// Mitsubishi GX Works2 project: onwork_noon   PLC: FX3G

// global labels: Global1
VAR_GLOBAL
  start_machineA AT X010 : BOOL;
  Touch_Sen AT M1 : BOOL;
  stop_machineA AT X005 : BOOL;
  Sen_Camera AT M2 : BOOL;
  Sen_30 AT X001 : BOOL;
  Ziluf_on AT Y004 : BOOL;
  Sen_15 AT X002 : BOOL;
  helpA AT M3 : BOOL;
  REG_InvetoryBiscuits AT D1102 : REAL;
END_VAR
VAR_GLOBAL CONSTANT
  Const_Biscuits : REAL := 6;
END_VAR
VAR_GLOBAL
  REG_Ziluf AT D1110 : REAL;
  REG_InvetoryCream AT D1104 : REAL;
END_VAR
VAR_GLOBAL CONSTANT
  Const_Cream : REAL := 300;
  Const_Zero : REAL;
  Const_InitInventoryBiscuits : REAL := 12;
  Const_InitInventoryCream : REAL := 600;
END_VAR
VAR_GLOBAL
  Sw_7_StartDay AT X007 : BOOL;
  M_TurnOffAll AT M7 : BOOL;
  Li_7_Day AT Y007 : BOOL;
  M_StartBlinking AT M8 : BOOL;
  Light_Generator AT M9 : BOOL;
  TC_BLINK_1 AT TC1 : BOOL;
  TS_BLINK_1 AT TS1 : BOOL;
  M_Blinking_Light1 AT M200 : BOOL;
  TC_BLINK_2 AT TC2 : BOOL;
END_VAR
VAR_GLOBAL CONSTANT
  CONSTANT3_word : INT := 3;
END_VAR
VAR_GLOBAL
  TS_BLINK_2 AT TS2 : BOOL;
  M_Blinking_Light2 AT M201 : BOOL;
  REG_InvetoryChocolate AT D1106 : REAL;
END_VAR
VAR_GLOBAL CONSTANT
  Const_Chocolate : REAL := 240;
END_VAR
VAR_GLOBAL
  M_InvetoryBiscuits AT M10 : BOOL;
  M_InvetoryCream AT M11 : BOOL;
  M_InvetoryChocolate AT M12 : BOOL;
  M_canStartDay AT M13 : BOOL;
  Current_in_process AT D1118 : REAL;
  Ziluf_timer AT TC0 : BOOL;
  TimerZiluf AT TC3 : BOOL;
END_VAR
VAR_GLOBAL CONSTANT
  TwoSeconds : INT := 20;
  SixSeconds : INT := 60;
END_VAR
VAR_GLOBAL
  TC_Shinua AT TC5 : BOOL;
END_VAR
VAR_GLOBAL CONSTANT
  FourSeconds : INT := 40;
END_VAR
VAR_GLOBAL
  TS_Shinua AT TS5 : BOOL;
  Sw_CreamToZiluf AT X011 : BOOL;
  TS_Ziluf AT TS3 : BOOL;
  TransportLight0 AT Y000 : BOOL;
  TrS1 AT Y001 : BOOL;
  TC_CloseDayTimer AT TC12 : BOOL;
END_VAR
VAR_GLOBAL CONSTANT
  ThreeSeconds : INT := 30;
END_VAR
VAR_GLOBAL
  TS_CloseDayTimer AT TS12 : BOOL;
  Ziluf_is_empty AT M22 : BOOL;
  Current_is_empty AT M24 : BOOL;
  Ziluf_is_full AT M23 : BOOL;
END_VAR
VAR_GLOBAL CONSTANT
  Const_CreamInit : REAL := 600;
  Const_ChocolateInit : REAL := 1000;
  Const_BiscuitsInit : REAL := 20;
END_VAR
VAR_GLOBAL
  input_pulse AT X006 : BOOL;
  analon_input_1 AT D8280 : INT;
  analog_input_val AT D1150 : REAL;
END_VAR
VAR_GLOBAL CONSTANT
  val1_analog_input_1 : REAL := 419;
END_VAR
VAR_GLOBAL
  frosting_type AT D4000 : REAL;
END_VAR
VAR_GLOBAL CONSTANT
  val1 : REAL := 1;
END_VAR
VAR_GLOBAL
  greater_than_1 AT M20 : BOOL;
END_VAR
VAR_GLOBAL CONSTANT
  val5 : REAL := 5;
END_VAR
VAR_GLOBAL
  less_than_5 AT M57 : BOOL;
  in_process AT TS7 : BOOL;
  double_frosting AT M32 : BOOL;
  regular_frosting AT M30 : BOOL;
END_VAR
VAR_GLOBAL CONSTANT
  val6 : REAL := 6;
END_VAR
VAR_GLOBAL
  greater_than_6 AT M25 : BOOL;
END_VAR
VAR_GLOBAL CONSTANT
  val10 : REAL := 10;
END_VAR
VAR_GLOBAL
  less_than_10 AT M27 : BOOL;
END_VAR
VAR_GLOBAL CONSTANT
  val120 : REAL := 120;
END_VAR
VAR_GLOBAL
  REG_immersion_tank AT D6500 : REAL;
END_VAR
VAR_GLOBAL CONSTANT
  val240 : REAL := 240;
END_VAR
VAR_GLOBAL
  frosting_timer AT TC7 : BOOL;
END_VAR
VAR_GLOBAL CONSTANT
  val0 : REAL;
  five_sec : INT := 5;
END_VAR
VAR_GLOBAL
  frosting_light AT Y003 : BOOL;
  error AT Y005 : BOOL;
  REG_CHECK AT D7000 : REAL;
  TimerZiluf_indicator AT TS3 : BOOL;
  pack_krembo AT X000 : BOOL;
  REG_done_indevidual_k_platform AT D3002 : REAL;
  almost_done_packing_platform AT Y002 : BOOL;
  REG_done_krembo_total AT D2222 : REAL;
END_VAR
VAR_GLOBAL CONSTANT
  const40 : REAL := 40;
END_VAR
VAR_GLOBAL
  VALUE_OUTPUT_ANALOG AT D2121 : REAL;
  value_analog_show_screen_REALLY AT D8282 : INT;
  done3 AT M14 : BOOL;
  start_pack AT M40 : BOOL;
  light_timer2_off AT TS2 : BOOL;
  light_timer1_off AT TS1 : BOOL;
  end_successfully AT M15 : BOOL;
  done4 AT M39 : BOOL;
  added_done_packed AT M45 : BOOL;
  timer_reset AT M42 : BOOL;
  light_counter AT CC10 : BOOL;
END_VAR
VAR_GLOBAL CONSTANT
  val3 : INT := 3;
END_VAR
VAR_GLOBAL
  light_counter_val AT CN10 : INT;
  need_flash AT M35 : BOOL;
END_VAR
VAR_GLOBAL CONSTANT
  val1_word : INT := 1;
END_VAR
VAR_GLOBAL
  supply_end AT M21 : BOOL;
  blink_end1 AT M47 : BOOL;
  no_supply_timer AT TC9 : BOOL;
END_VAR
VAR_GLOBAL CONSTANT
  three_sec : INT := 30;
END_VAR
VAR_GLOBAL
  TS_nosupply_timer AT TS9 : BOOL;
  M49_Y7 AT M49 : BOOL;
  tm_nosupply2 AT TC11 : BOOL;
  TS2_nosup AT TS11 : BOOL;
  M51_offM49 AT M51 : BOOL;
  final_tm AT TC15 : BOOL;
  final_tm_indecator AT TS15 : BOOL;
  blink_indecator AT M55 : BOOL;
END_VAR
VAR_GLOBAL CONSTANT
  five_sec_frosting : INT := 50;
END_VAR
VAR_GLOBAL
  not_enough_krembo AT M13 : BOOL;
END_VAR

// task Task_01 (event TRUE, interval 0, priority 31): POU_01

PROGRAM POU_01
VAR
  TransportLight1 : BOOL;
END_VAR
(* structured ladder/FBD written out as ST: instructions are called as NAME(EN, inputs, outputs); _pN, _eN, _tN stand for wires *)
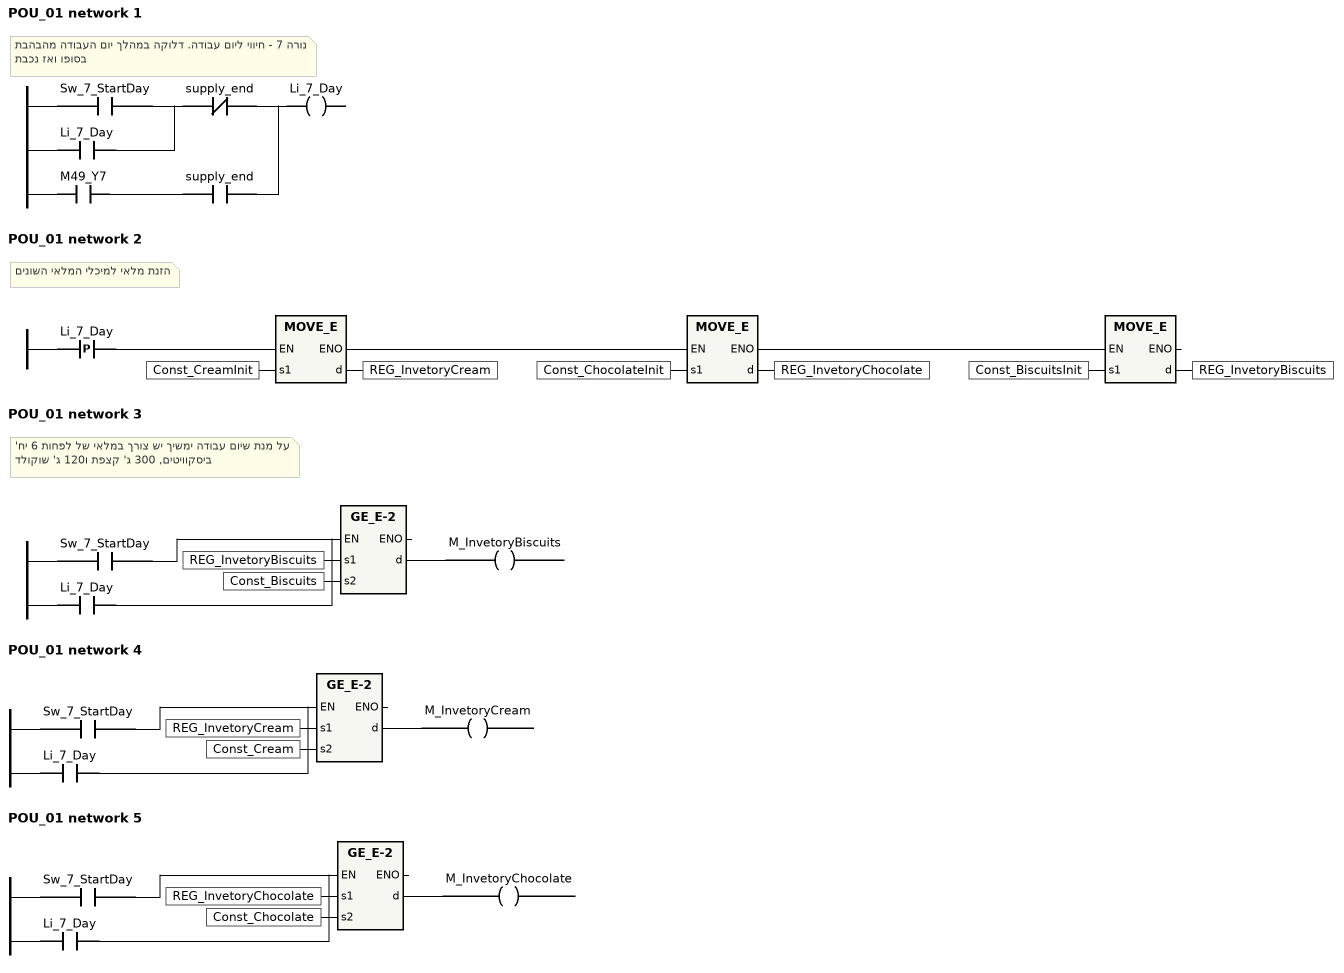
(* network 1 *)
(* נורה 7 - חיווי ליום עבודה. דלוקה במהלך יום העבודה מהבהבת בסופו ואז נכבת *)
Li_7_Day := ((Sw_7_StartDay OR Li_7_Day) AND NOT supply_end) OR (M49_Y7 AND supply_end);
(* network 2 *)
(* הזנת מלאי למיכלי המלאי השונים *)
_e1 := MOVE_E(LDP(TRUE, Li_7_Day), Const_CreamInit, REG_InvetoryCream);
_e2 := MOVE_E(_e1, Const_ChocolateInit, REG_InvetoryChocolate);
MOVE_E(_e2, Const_BiscuitsInit, REG_InvetoryBiscuits);
(* network 3 *)
(* על מנת שיום עבודה ימשיך יש צורך במלאי של לפחות 6 יח' ביסקוויטים, 300 ג' קצפת ו120 ג' שוקולד *)
GE_E(Sw_7_StartDay OR Li_7_Day, REG_InvetoryBiscuits, Const_Biscuits, _t1);
M_InvetoryBiscuits := _t1;
(* network 4 *)
GE_E(Sw_7_StartDay OR Li_7_Day, REG_InvetoryCream, Const_Cream, _t1);
M_InvetoryCream := _t1;
(* network 5 *)
GE_E(Sw_7_StartDay OR Li_7_Day, REG_InvetoryChocolate, Const_Chocolate, _t1);
M_InvetoryChocolate := _t1;
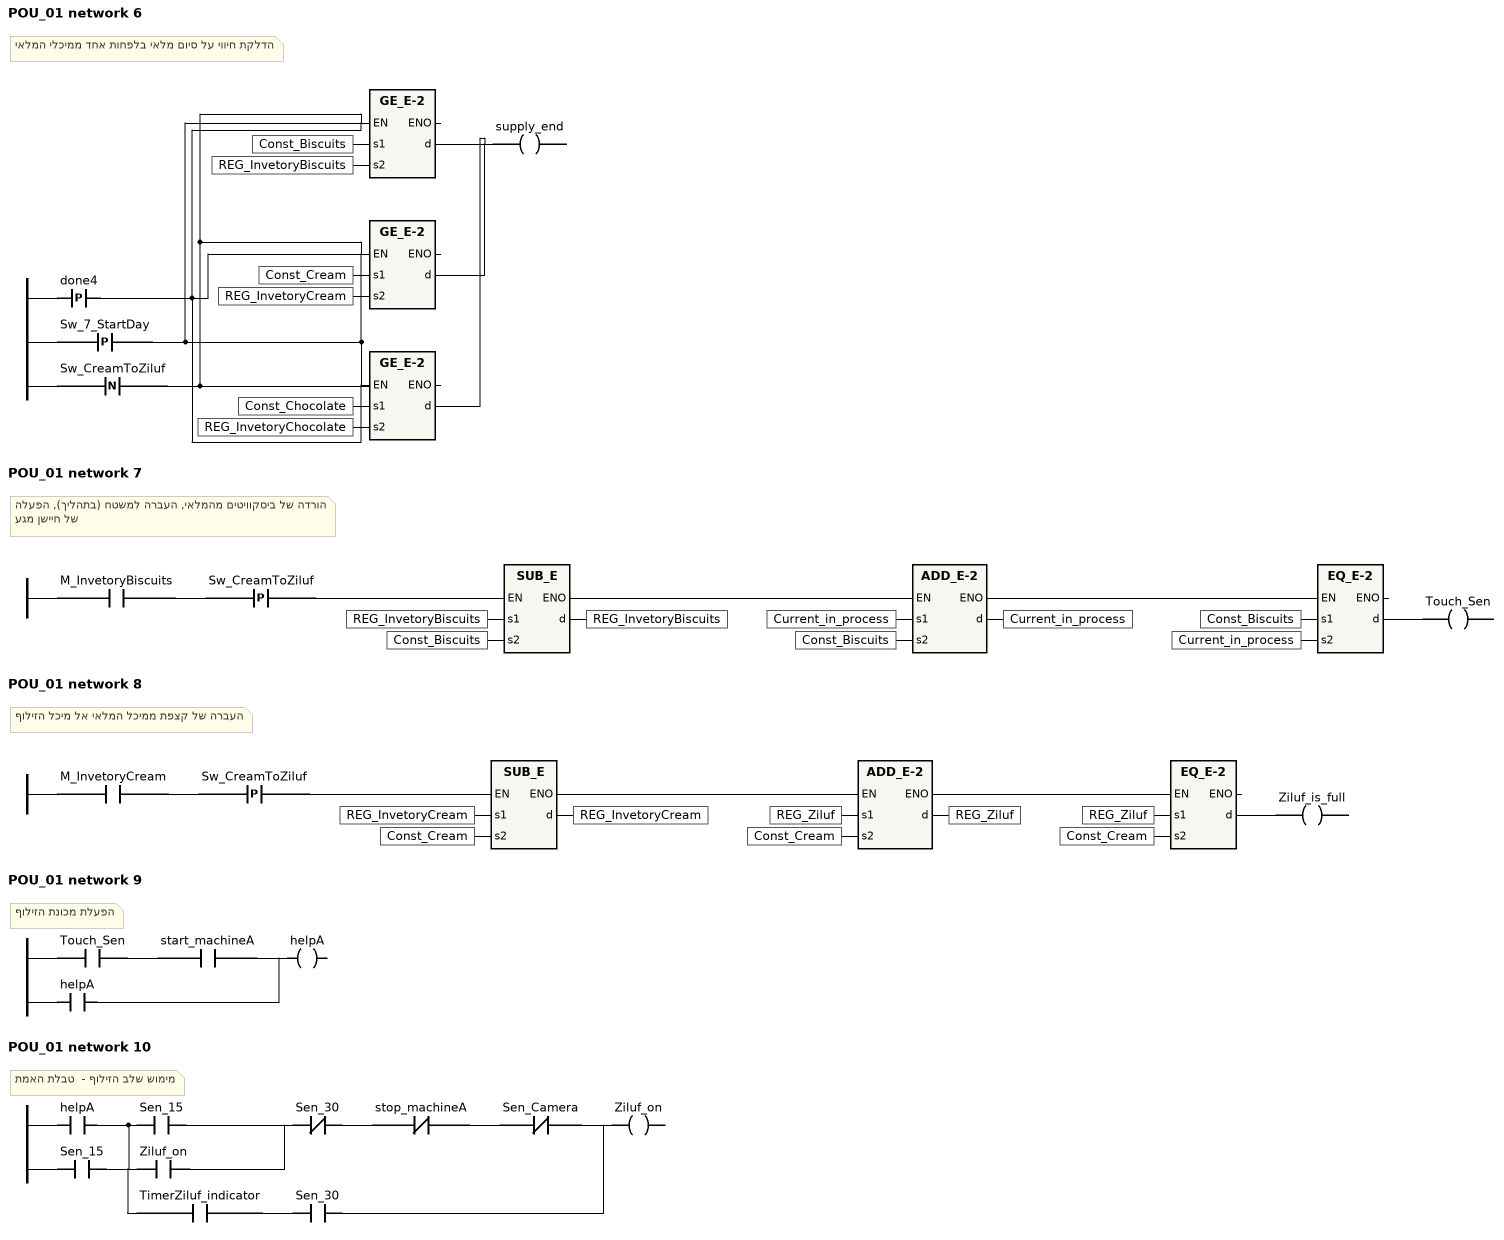
(* network 6 *)
(* הדלקת חיווי על סיום מלאי בלפחות אחד ממיכלי המלאי *)
_p1 := LDP(TRUE, done4) OR LDP(TRUE, Sw_7_StartDay) OR LDF(TRUE, Sw_CreamToZiluf);
GE_E(_p1, Const_Biscuits, REG_InvetoryBiscuits, _t2);
GE_E(_p1, Const_Cream, REG_InvetoryCream, _t3);
GE_E(_p1, Const_Chocolate, REG_InvetoryChocolate, _t4);
supply_end := _t2 OR _t3 OR _t4;
(* network 7 *)
(* הורדה של ביסקוויטים מהמלאי, העברה למשטח (בתהליך), הפעלה של חיישן מגע *)
_e1 := SUB_E(M_InvetoryBiscuits AND LDP(TRUE, Sw_CreamToZiluf), REG_InvetoryBiscuits, Const_Biscuits, REG_InvetoryBiscuits);
_e2 := ADD_E(_e1, Current_in_process, Const_Biscuits, Current_in_process);
EQ_E(_e2, Const_Biscuits, Current_in_process, _t3);
Touch_Sen := _t3;
(* network 8 *)
(* העברה של קצפת ממיכל המלאי אל מיכל הזילוף *)
_e1 := SUB_E(M_InvetoryCream AND LDP(TRUE, Sw_CreamToZiluf), REG_InvetoryCream, Const_Cream, REG_InvetoryCream);
_e2 := ADD_E(_e1, REG_Ziluf, Const_Cream, REG_Ziluf);
EQ_E(_e2, REG_Ziluf, Const_Cream, _t3);
Ziluf_is_full := _t3;
(* network 9 *)
(* הפעלת מכונת הזילוף *)
helpA := (Touch_Sen AND start_machineA) OR helpA;
(* network 10 *)
(* מימוש שלב הזילוף -  טבלת האמת *)
Ziluf_on := (((((helpA AND Sen_15) OR (helpA AND Ziluf_on)) AND NOT Sen_30) AND NOT stop_machineA) AND NOT Sen_Camera) OR (Sen_15 AND TimerZiluf_indicator AND Sen_30);
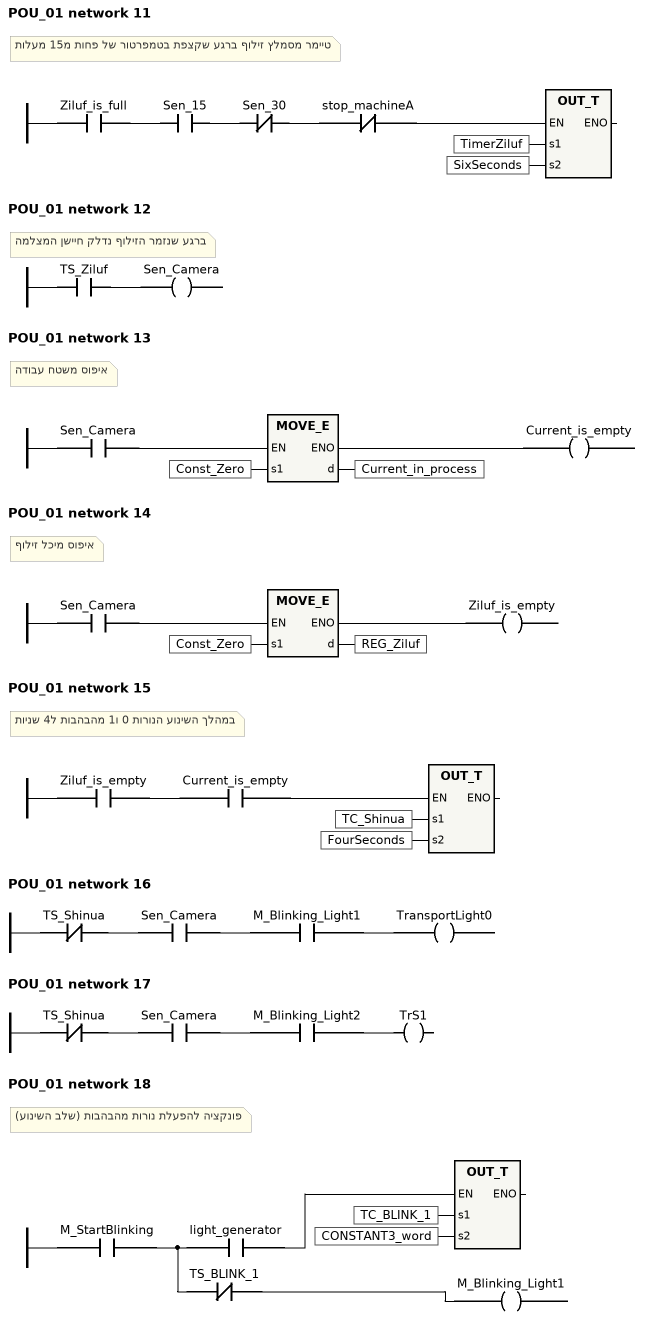
(* network 11 *)
(* טיימר מסמלץ זילוף ברגע שקצפת בטמפרטור של פחות מ15 מעלות *)
OUT_T(Ziluf_is_full AND Sen_15 AND NOT Sen_30 AND NOT stop_machineA, TimerZiluf, SixSeconds);
(* network 12 *)
(* ברגע שנזמר הזילוף נדלק חיישן המצלמה *)
Sen_Camera := TS_Ziluf;
(* network 13 *)
(* איפוס משטח עבודה *)
_e1 := MOVE_E(Sen_Camera, Const_Zero, Current_in_process);
Current_is_empty := _e1;
(* network 14 *)
(* איפוס מיכל זילוף *)
_e1 := MOVE_E(Sen_Camera, Const_Zero, REG_Ziluf);
Ziluf_is_empty := _e1;
(* network 15 *)
(* במהלך השינוע הנורות 0 ו1 מהבהבות ל4 שניות *)
OUT_T(Ziluf_is_empty AND Current_is_empty, TC_Shinua, FourSeconds);
(* network 16 *)
TransportLight0 := NOT TS_Shinua AND Sen_Camera AND M_Blinking_Light1;
(* network 17 *)
TrS1 := NOT TS_Shinua AND Sen_Camera AND M_Blinking_Light2;
(* network 18 *)
(* פונקציה להפעלת נורות מהבהבות (שלב השינוע) *)
OUT_T(M_StartBlinking AND light_generator, TC_BLINK_1, CONSTANT3_word);
M_Blinking_Light1 := M_StartBlinking AND NOT TS_BLINK_1;
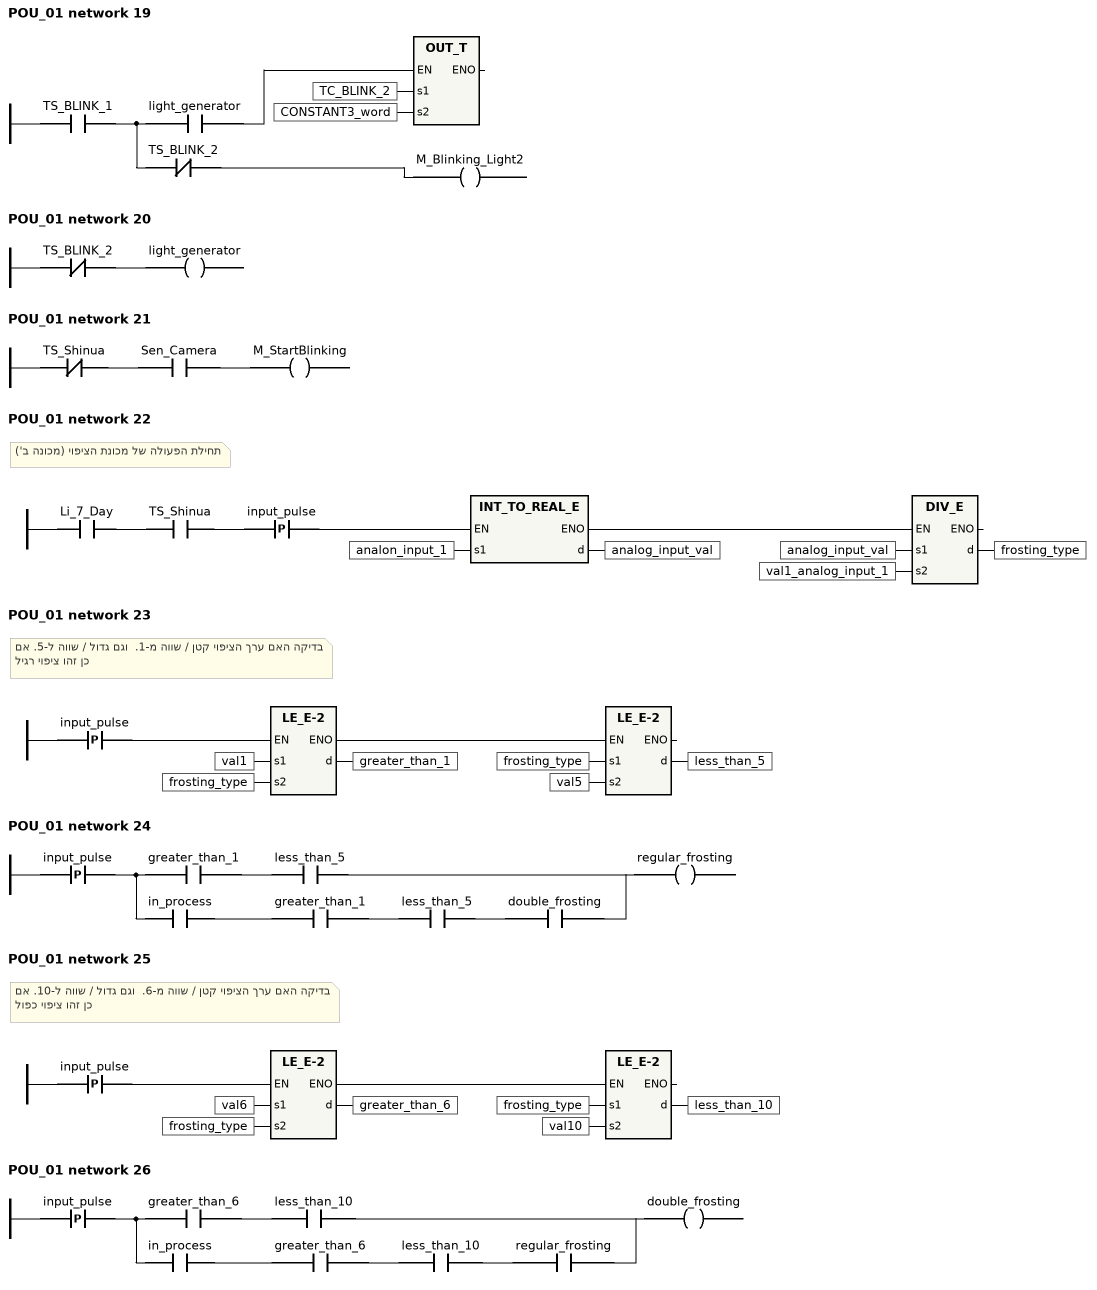
(* network 19 *)
OUT_T(TS_BLINK_1 AND light_generator, TC_BLINK_2, CONSTANT3_word);
M_Blinking_Light2 := TS_BLINK_1 AND NOT TS_BLINK_2;
(* network 20 *)
light_generator := NOT TS_BLINK_2;
(* network 21 *)
M_StartBlinking := NOT TS_Shinua AND Sen_Camera;
(* network 22 *)
(* תחילת הפעולה של מכונת הציפוי (מכונה ב') *)
_e1 := INT_TO_REAL_E(Li_7_Day AND TS_Shinua AND LDP(TRUE, input_pulse), analon_input_1, analog_input_val);
DIV_E(_e1, analog_input_val, val1_analog_input_1, frosting_type);
(* network 23 *)
(* בדיקה האם ערך הציפוי קטן / שווה מ-1.  וגם גדול / שווה ל-5. אם כן זהו ציפוי רגיל *)
_e1 := LE_E(LDP(TRUE, input_pulse), val1, frosting_type, greater_than_1);
LE_E(_e1, frosting_type, val5, less_than_5);
(* network 24 *)
_p1 := LDP(TRUE, input_pulse);
regular_frosting := (_p1 AND greater_than_1 AND less_than_5) OR (_p1 AND in_process AND greater_than_1 AND less_than_5 AND double_frosting);
(* network 25 *)
(* בדיקה האם ערך הציפוי קטן / שווה מ-6.  וגם גדול / שווה ל-10. אם כן זהו ציפוי כפול *)
_e1 := LE_E(LDP(TRUE, input_pulse), val6, frosting_type, greater_than_6);
LE_E(_e1, frosting_type, val10, less_than_10);
(* network 26 *)
_p1 := LDP(TRUE, input_pulse);
double_frosting := (_p1 AND greater_than_6 AND less_than_10) OR (_p1 AND in_process AND greater_than_6 AND less_than_10 AND regular_frosting);
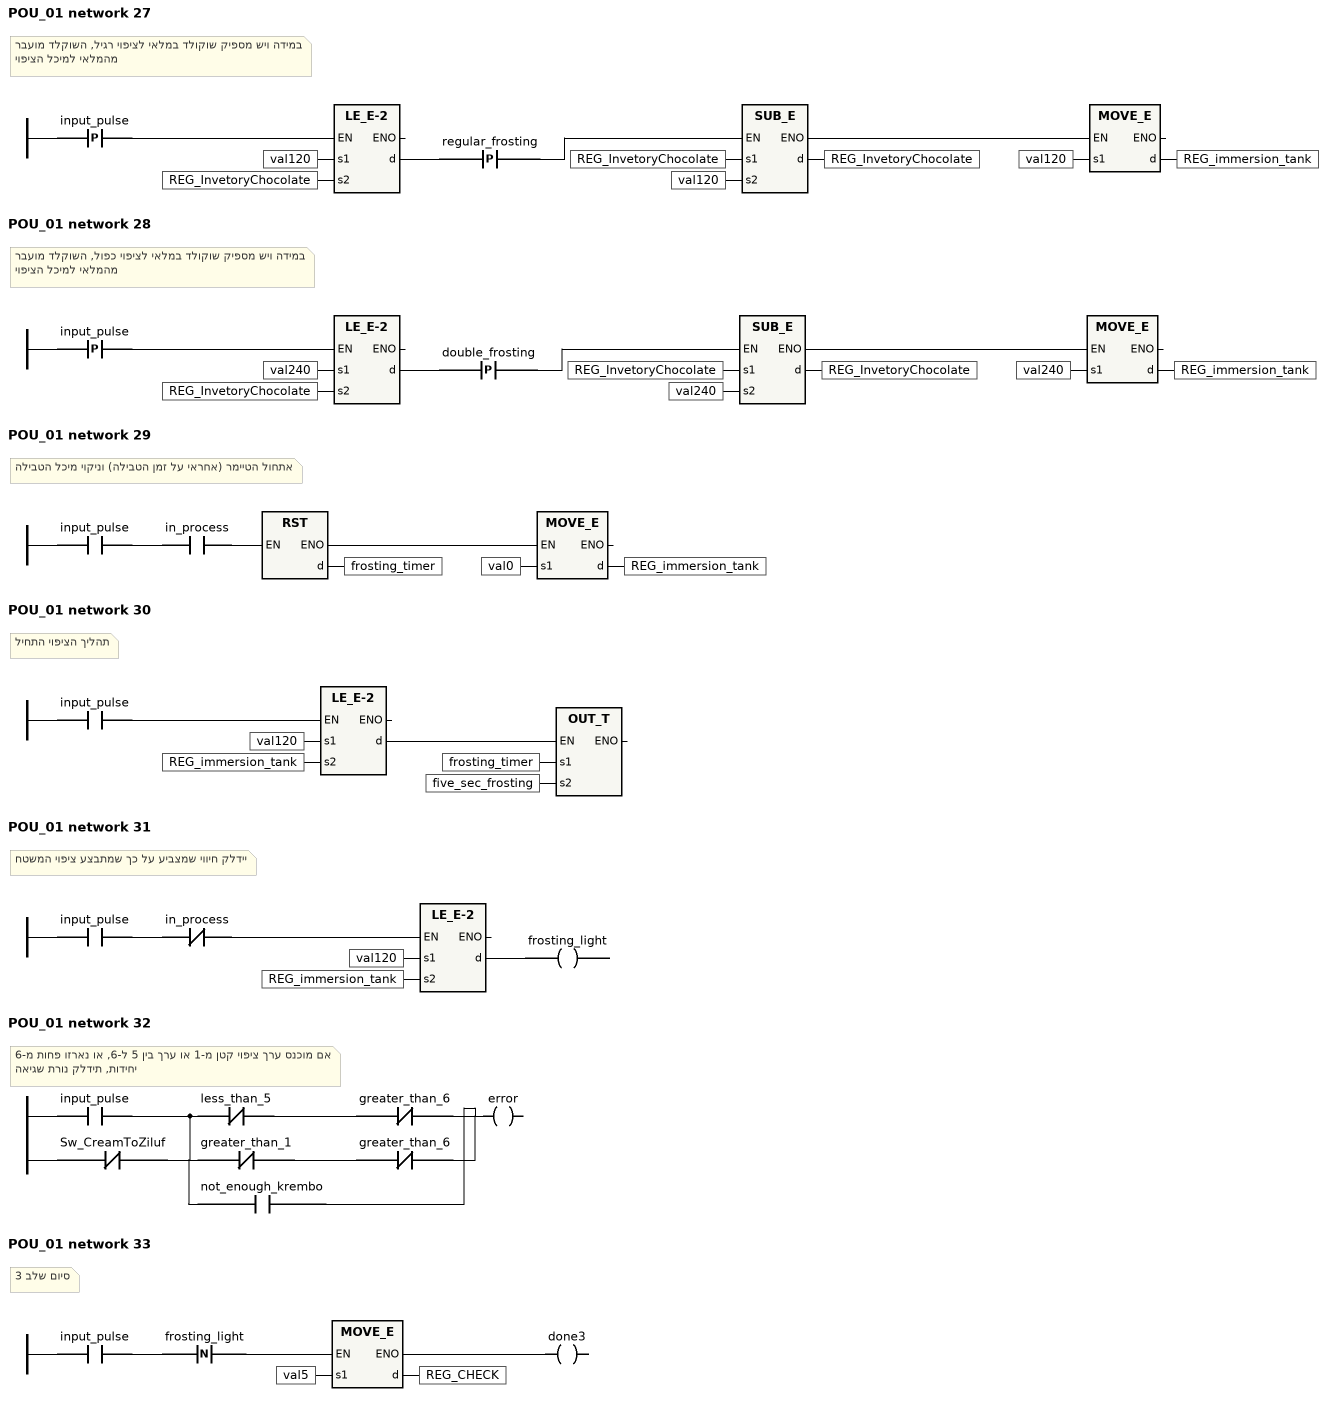
(* network 27 *)
(* במידה ויש מספיק שוקולד במלאי לציפוי רגיל, השוקלד מועבר מהמלאי למיכל הציפוי *)
LE_E(LDP(TRUE, input_pulse), val120, REG_InvetoryChocolate, _t1);
_e2 := SUB_E(_t1 AND LDP(TRUE, regular_frosting), REG_InvetoryChocolate, val120, REG_InvetoryChocolate);
MOVE_E(_e2, val120, REG_immersion_tank);
(* network 28 *)
(* במידה ויש מספיק שוקולד במלאי לציפוי כפול, השוקלד מועבר מהמלאי למיכל הציפוי *)
LE_E(LDP(TRUE, input_pulse), val240, REG_InvetoryChocolate, _t1);
_e2 := SUB_E(_t1 AND LDP(TRUE, double_frosting), REG_InvetoryChocolate, val240, REG_InvetoryChocolate);
MOVE_E(_e2, val240, REG_immersion_tank);
(* network 29 *)
(* אתחול הטיימר (אחראי על זמן הטבילה) וניקוי מיכל הטבילה *)
_e1 := RST(input_pulse AND in_process, frosting_timer);
MOVE_E(_e1, val0, REG_immersion_tank);
(* network 30 *)
(* תהליך הציפוי התחיל *)
LE_E(input_pulse, val120, REG_immersion_tank, _t1);
OUT_T(_t1, frosting_timer, five_sec_frosting);
(* network 31 *)
(* יידלק חיווי שמצביע על כך שמתבצע ציפוי המשטח *)
LE_E(input_pulse AND NOT in_process, val120, REG_immersion_tank, _t1);
frosting_light := _t1;
(* network 32 *)
(* אם מוכנס ערך ציפוי קטן מ-1 או ערך בין 5 ל-6, או נארזו פחות מ-6 יחידות, תידלק נורת שגיאה *)
error := (input_pulse AND NOT less_than_5 AND NOT greater_than_6) OR (input_pulse AND NOT greater_than_1 AND NOT greater_than_6) OR (NOT Sw_CreamToZiluf AND not_enough_krembo);
(* network 33 *)
(* סיום שלב 3 *)
_e1 := MOVE_E(input_pulse AND LDF(TRUE, frosting_light), val5, REG_CHECK);
done3 := _e1;
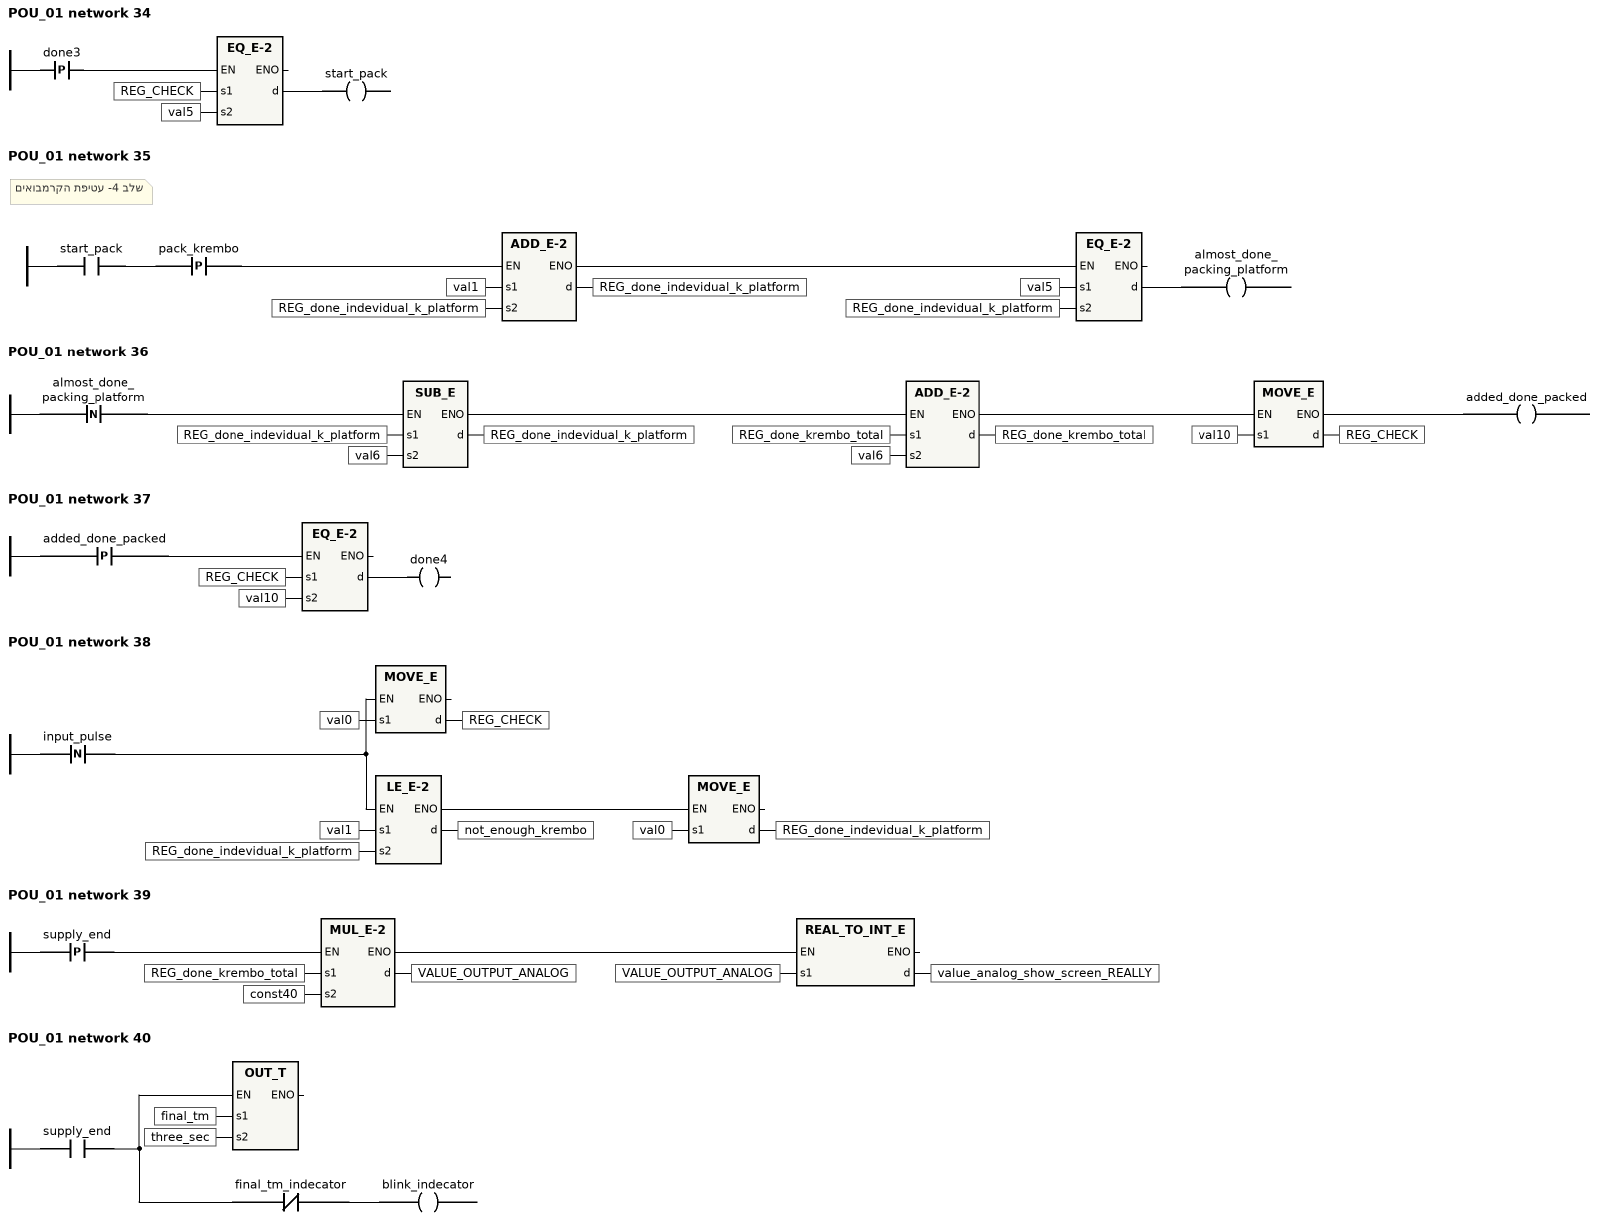
(* network 34 *)
EQ_E(LDP(TRUE, done3), REG_CHECK, val5, _t1);
start_pack := _t1;
(* network 35 *)
(* שלב 4- עטיפת הקרמבואים *)
_e1 := ADD_E(start_pack AND LDP(TRUE, pack_krembo), val1, REG_done_indevidual_k_platform, REG_done_indevidual_k_platform);
EQ_E(_e1, val5, REG_done_indevidual_k_platform, _t2);
almost_done_packing_platform := _t2;
(* network 36 *)
_e1 := SUB_E(LDF(TRUE, almost_done_packing_platform), REG_done_indevidual_k_platform, val6, REG_done_indevidual_k_platform);
_e2 := ADD_E(_e1, REG_done_krembo_total, val6, REG_done_krembo_total);
_e3 := MOVE_E(_e2, val10, REG_CHECK);
added_done_packed := _e3;
(* network 37 *)
EQ_E(LDP(TRUE, added_done_packed), REG_CHECK, val10, _t1);
done4 := _t1;
(* network 38 *)
_p1 := LDF(TRUE, input_pulse);
MOVE_E(_p1, val0, REG_CHECK);
_e2 := LE_E(_p1, val1, REG_done_indevidual_k_platform, not_enough_krembo);
MOVE_E(_e2, val0, REG_done_indevidual_k_platform);
(* network 39 *)
_e1 := MUL_E(LDP(TRUE, supply_end), REG_done_krembo_total, const40, VALUE_OUTPUT_ANALOG);
REAL_TO_INT_E(_e1, VALUE_OUTPUT_ANALOG, value_analog_show_screen_REALLY);
(* network 40 *)
OUT_T(supply_end, final_tm, three_sec);
blink_indecator := supply_end AND NOT final_tm_indecator;
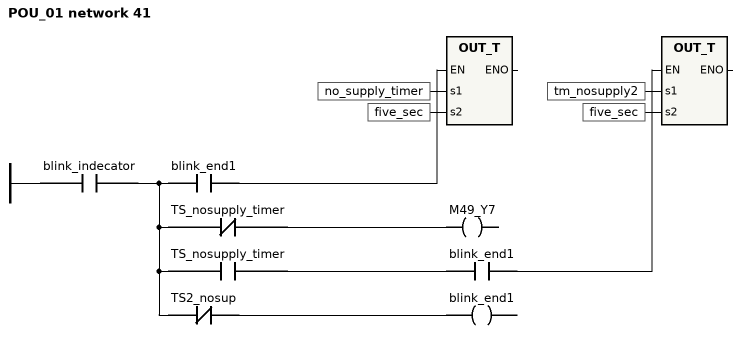
(* network 41 *)
OUT_T(blink_indecator AND blink_end1, no_supply_timer, five_sec);
M49_Y7 := blink_indecator AND NOT TS_nosupply_timer;
OUT_T(blink_indecator AND TS_nosupply_timer AND blink_end1, tm_nosupply2, five_sec);
blink_end1 := blink_indecator AND NOT TS2_nosup;
END_PROGRAM
